// TIA Portal V17 export
// export: Created 2025-05-22T06:00:34.8256943Z, ExportSetting WithDefaults, DisplayName Totally Integrated Automation Portal, DisplayVersion V17 Update 8, DisplayName TIA Portal Openness, DisplayVersion V17 Update 8, DisplayName TIA Portal Version Control Interface, DisplayVersion V17, DisplayName SINAMICS Startdrive Advanced, DisplayVersion V17 SP2, DisplayName SINAMICS Startdrive G110M, G120, G120C, G120D, G120P, G115D, DisplayVersion V17 SP2, DisplayName SINAMICS Startdrive G130, G150, S120, S150, SINAMICS MV, S210, DisplayVersion V17 SP2, DisplayName STEP 7 Professional, DisplayVersion V17 Update 8, DisplayName SINUMERIK ONE STEP 7 Toolbox, DisplayVersion V17 Update 12, DisplayName SINUMERIK ONE PLC Basic Program Plus, DisplayVersion V17 Update 12, DisplayName SINUMERIK 840D sl STEP 7 Toolbox, DisplayVersion V17 Update 12, DisplayName STEP 7 Safety, DisplayVersion V17 Update 6, DisplayName WinCC Advanced, DisplayVersion V17 Update 8
FUNCTION "FC6692_SAFETY_BRAKE_Z13" : Void   // FC6692, LAD
{ S7_Optimized_Access := 'FALSE' }
AUTHOR : ETXETAR
VERSION : 1.0
// stored: AutoNumber false, IsIECCheckEnabled false, SetENOAutomatically false, UDAEnableTagReadback false
   VAR_TEMP   // added for the SCL form of the ladder/FBD networks
      _w1 : Bool;
   END_VAR
BEGIN

REGION Network 1: CALL FB6600 SAFETY BRAKE Y1 AXIS / SAFETY BRAKE Y1 AXIS - 01R
   // 2#0000_0001 OPTIONS 0 BIT 0 MAINTENANCE SENSORS OPTION
   // 2#0000_0010 OPTIONS 0 BIT 1 SPARE OPTION
   // 2#0000_0100 OPTIONS 0 BIT 2 SPARE OPTION
   // 2#0000_1000 OPTIONS 0 BIT 3 SPARE OPTION
   // 2#0001_0000 OPTIONS 0 BIT 4 SPARE OPTION
   // 2#0010_0000 OPTIONS 0 BIT 5 SPARE OPTION
   // 2#0100_0000 OPTIONS 0 BIT 6 SPARE OPTION
   // 2#1000_0000 OPTIONS 0 BIT 7 SPARE OPTION
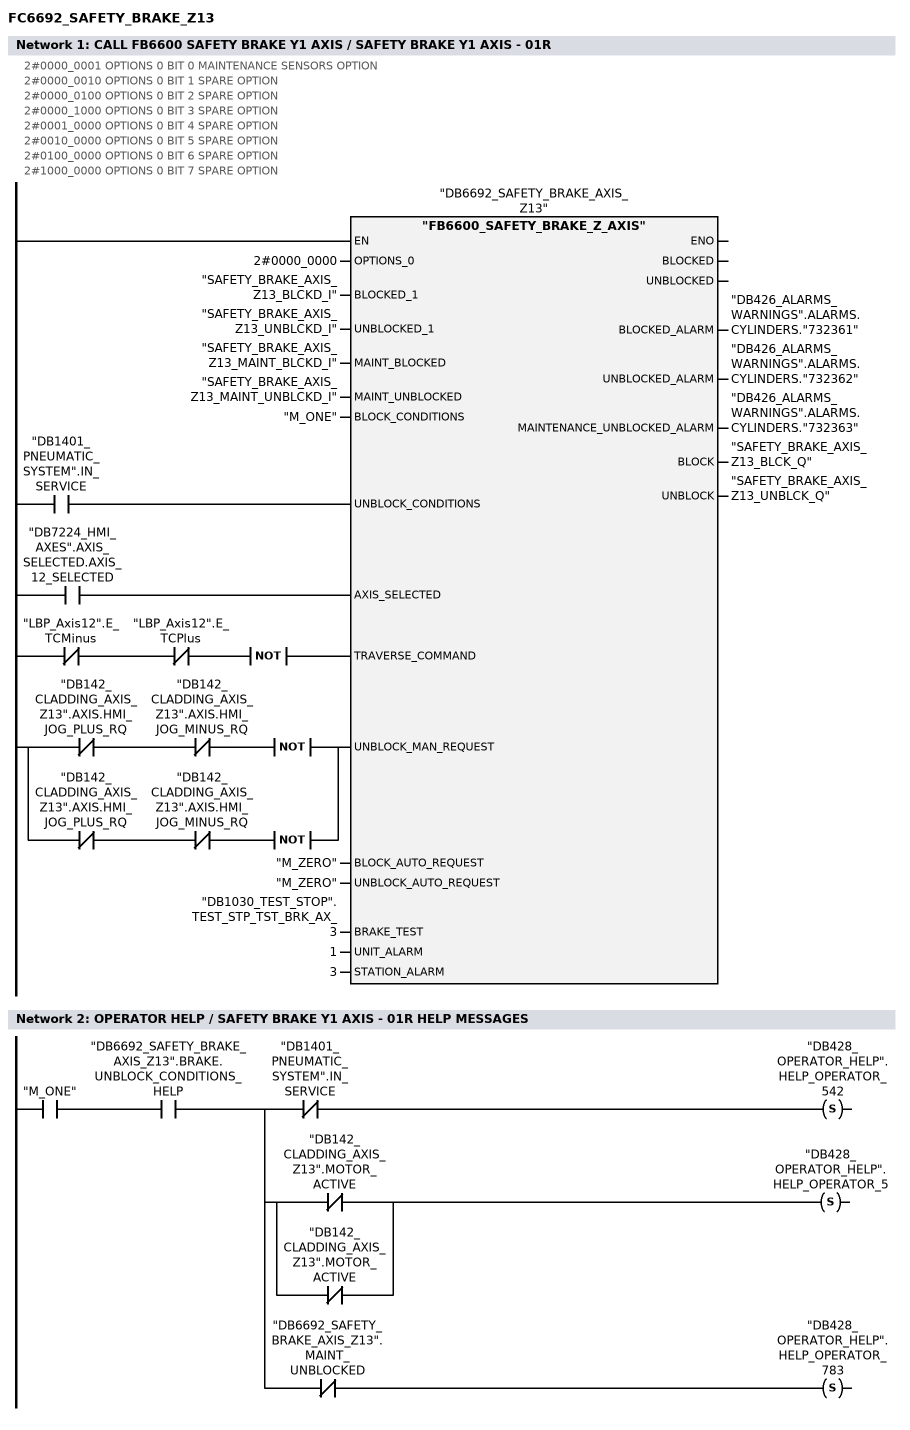
   RUNG wire#powerrail
      "DB6692_SAFETY_BRAKE_AXIS_Z13"(UNBLOCK_CONDITIONS := wire#w1, AXIS_SELECTED := wire#w2, TRAVERSE_COMMAND := wire#w3, UNBLOCK_MAN_REQUEST := wire#w4, OPTIONS_0 := 2#0000_0000, BLOCKED_1 := "SAFETY_BRAKE_AXIS_Z13_BLCKD_I", UNBLOCKED_1 := "SAFETY_BRAKE_AXIS_Z13_UNBLCKD_I", MAINT_BLOCKED := "SAFETY_BRAKE_AXIS_Z13_MAINT_BLCKD_I", MAINT_UNBLOCKED := "SAFETY_BRAKE_AXIS_Z13_MAINT_UNBLCKD_I", BLOCK_CONDITIONS := "M_ONE", BLOCK_AUTO_REQUEST := "M_ZERO", UNBLOCK_AUTO_REQUEST := "M_ZERO", BRAKE_TEST := "DB1030_TEST_STOP".TEST_STP_TST_BRK_AX_3, UNIT_ALARM := 1, STATION_ALARM := 3, BLOCKED =>, UNBLOCKED =>, BLOCKED_ALARM => "DB426_ALARMS_WARNINGS".ALARMS.CYLINDERS."732361", UNBLOCKED_ALARM => "DB426_ALARMS_WARNINGS".ALARMS.CYLINDERS."732362", MAINTENANCE_UNBLOCKED_ALARM => "DB426_ALARMS_WARNINGS".ALARMS.CYLINDERS."732363", BLOCK => "SAFETY_BRAKE_AXIS_Z13_BLCK_Q", UNBLOCK => "SAFETY_BRAKE_AXIS_Z13_UNBLCK_Q")
   END_RUNG
   RUNG wire#powerrail
      Contact( "DB1401_PNEUMATIC_SYSTEM".IN_SERVICE )
   END_RUNG wire#w1
   RUNG wire#powerrail
      Contact( "DB7224_HMI_AXES".AXIS_SELECTED.AXIS_12_SELECTED )
   END_RUNG wire#w2
   RUNG wire#powerrail
      I_Contact( "LBP_Axis12".E_TCMinus )
      I_Contact( "LBP_Axis12".E_TCPlus )
      Not()
   END_RUNG wire#w3
   RUNG wire#powerrail
      I_Contact( "DB142_CLADDING_AXIS_Z13".AXIS.HMI_JOG_PLUS_RQ )
      I_Contact( "DB142_CLADDING_AXIS_Z13".AXIS.HMI_JOG_MINUS_RQ )
      Not()
   END_RUNG wire#w4
   RUNG wire#powerrail
      I_Contact( "DB142_CLADDING_AXIS_Z13".AXIS.HMI_JOG_PLUS_RQ )
      I_Contact( "DB142_CLADDING_AXIS_Z13".AXIS.HMI_JOG_MINUS_RQ )
      Not()
   END_RUNG wire#w4
   // the same network as SCL:
   "DB6692_SAFETY_BRAKE_AXIS_Z13"(OPTIONS_0 := 2#0000_0000,   // "FB6600_SAFETY_BRAKE_Z_AXIS"
                           BLOCKED_1 := "SAFETY_BRAKE_AXIS_Z13_BLCKD_I",
                           UNBLOCKED_1 := "SAFETY_BRAKE_AXIS_Z13_UNBLCKD_I",
                           MAINT_BLOCKED := "SAFETY_BRAKE_AXIS_Z13_MAINT_BLCKD_I",
                           MAINT_UNBLOCKED := "SAFETY_BRAKE_AXIS_Z13_MAINT_UNBLCKD_I",
                           BLOCK_CONDITIONS := "M_ONE",
                           UNBLOCK_CONDITIONS := "DB1401_PNEUMATIC_SYSTEM".IN_SERVICE,
                           AXIS_SELECTED := "DB7224_HMI_AXES".AXIS_SELECTED.AXIS_12_SELECTED,
                           TRAVERSE_COMMAND := NOT (NOT "LBP_Axis12".E_TCMinus AND NOT "LBP_Axis12".E_TCPlus),
                           UNBLOCK_MAN_REQUEST := NOT (NOT "DB142_CLADDING_AXIS_Z13".AXIS.HMI_JOG_PLUS_RQ AND NOT "DB142_CLADDING_AXIS_Z13".AXIS.HMI_JOG_MINUS_RQ) OR NOT (NOT "DB142_CLADDING_AXIS_Z13".AXIS.HMI_JOG_PLUS_RQ AND NOT "DB142_CLADDING_AXIS_Z13".AXIS.HMI_JOG_MINUS_RQ),
                           BLOCK_AUTO_REQUEST := "M_ZERO",
                           UNBLOCK_AUTO_REQUEST := "M_ZERO",
                           BRAKE_TEST := "DB1030_TEST_STOP".TEST_STP_TST_BRK_AX_3,
                           UNIT_ALARM := 1,
                           STATION_ALARM := 3,
                           BLOCKED_ALARM => "DB426_ALARMS_WARNINGS".ALARMS.CYLINDERS."732361",
                           UNBLOCKED_ALARM => "DB426_ALARMS_WARNINGS".ALARMS.CYLINDERS."732362",
                           MAINTENANCE_UNBLOCKED_ALARM => "DB426_ALARMS_WARNINGS".ALARMS.CYLINDERS."732363",
                           BLOCK => "SAFETY_BRAKE_AXIS_Z13_BLCK_Q",
                           UNBLOCK => "SAFETY_BRAKE_AXIS_Z13_UNBLCK_Q");
END_REGION

REGION Network 2: OPERATOR HELP / SAFETY BRAKE Y1 AXIS - 01R HELP MESSAGES
   RUNG wire#powerrail
      Contact( "M_ONE" )
      Contact( "DB6692_SAFETY_BRAKE_AXIS_Z13".BRAKE.UNBLOCK_CONDITIONS_HELP )
      wire#w1
      I_Contact( "DB1401_PNEUMATIC_SYSTEM".IN_SERVICE )
      S_Coil( "DB428_OPERATOR_HELP".HELP_OPERATOR_542 )
   END_RUNG
   RUNG wire#w1
      I_Contact( "DB142_CLADDING_AXIS_Z13".MOTOR_ACTIVE )
      wire#w2
      S_Coil( "DB428_OPERATOR_HELP".HELP_OPERATOR_5 )
   END_RUNG
   RUNG wire#w1
      I_Contact( "DB142_CLADDING_AXIS_Z13".MOTOR_ACTIVE )
   END_RUNG wire#w2
   RUNG wire#w1
      I_Contact( "DB6692_SAFETY_BRAKE_AXIS_Z13".MAINT_UNBLOCKED )
      S_Coil( "DB428_OPERATOR_HELP".HELP_OPERATOR_783 )
   END_RUNG
   // the same network as SCL:
   #_w1 := "M_ONE" AND "DB6692_SAFETY_BRAKE_AXIS_Z13".BRAKE.UNBLOCK_CONDITIONS_HELP;
   IF #_w1 AND NOT "DB1401_PNEUMATIC_SYSTEM".IN_SERVICE THEN
       "DB428_OPERATOR_HELP".HELP_OPERATOR_542 := TRUE;
   END_IF;
   IF #_w1 AND (NOT "DB142_CLADDING_AXIS_Z13".MOTOR_ACTIVE OR NOT "DB142_CLADDING_AXIS_Z13".MOTOR_ACTIVE) THEN
       "DB428_OPERATOR_HELP".HELP_OPERATOR_5 := TRUE;
   END_IF;
   IF #_w1 AND NOT "DB6692_SAFETY_BRAKE_AXIS_Z13".MAINT_UNBLOCKED THEN
       "DB428_OPERATOR_HELP".HELP_OPERATOR_783 := TRUE;
   END_IF;
END_REGION
END_FUNCTION
